PROGRAM MAIN
VAR
	fastChain: TestAwaitChainFast;
	normalChain: TestAwaitChainNormal;
	postChain: TestPostLogChain;
END_VAR

fastChain();
normalChain();
postChain();

END_PROGRAM

(* stored: Version 1.1.0.1, ProductVersion 3.1.4024.12
   POU MAIN: Id {f3fedbc9-a740-4747-9cb3-fa9102cc0759}, SpecialFunc None *)
